// TIA Portal V19 export
DATA_BLOCK "HmiInterface"   // DB63
// stored: Access Published, MemoryReserve 100, Namespace Unit2.EM2
   VAR
      em : "LAF_typeEmInterface";
      jobs : "LAF_typeJobsInterface";
      sequence : "LAF_typeSequenceInterface";
      cm1Vfd206 : "LEXCHANGETRAY_typeRollerVfdInterface";
      cm2TrayLiftingCylinder { S7_SetPoint := 'True'} : "LBC_Simple_typeTwoWayActuatorInterface";
      cm3CellLiftingCylinder { S7_SetPoint := 'True'} : "LBC_Simple_typeTwoWayActuatorInterface";
      cm4PositioningPinCylinder { S7_SetPoint := 'True'} : "LBC_Simple_typeTwoWayActuatorInterface";
      cm5AxisControl { S7_SetPoint := 'True'} : "LBC_typeAxisSimpleControlInterface_1";
      cm6SignalTM { S7_SetPoint := 'True'} : "LEXCHANGETRAY_typeConstraintRollerIoSignalInterface";
      cm7Pc { S7_SetPoint := 'True'} : "LEXCHANGETRAY_typePc_Interface";
      cm8Scanner { S7_SetPoint := 'True'} : "LEXCHANGETRAY_typeSR1000Interface";
      em2Parameters : "LAF_typeConstraintRollerEm2ParametersInterface";
   END_VAR
BEGIN
END_DATA_BLOCK
